TYPE ST_Result :
STRUCT
	total		: REAL;
	energy		: REAL;
	tax			: REAL;
	startsAt	: STRING;
	level		: STRING;
END_STRUCT
END_TYPE

(* stored: Version 1.1.0.1, ProductVersion 3.1.4024.12
   DUT ST_Result: Id {6ddf8eb2-cd00-48a6-a971-888b44c92d5f} *)
